(*********************************** G.D S.p.A. - Technical Department ***********************************
============= PROGRAM INFO ============
FOLDER:             TBD
MACHINES INVOLVED:  TBD 

============= DESCRIPTION =============
csp machine declaration

============= REVISIONS ===============
Date		Version	 	Author      	Description             
----------	-------		------------  	--------------------------------------------
2019/04/05 	0000.00	 	M.Grasso		Creation of the PRG

**********************************************************************************************************)
(*$R process_ref := prc; $*)
PROGRAM csp_case_feed_kinematic_tilt
VAR
		
	prc:												process;
	prc_path:											STRING;
	
	axis:												axis;
	axis_actual_position:								LREAL;
	
	fsm_enable_condition:								BOOL := FALSE;
	fsm_next_status:									csp_case_feed_kinematic_status_enum;
	fsm_status:											csp_case_feed_kinematic_status_enum;
	debug_state_machine:								BOOL := FALSE;
	debug_state_machine_one_step:						BOOL := FALSE;	
	
	in_accu_safe_pos:                                   BOOL := FALSE;
    accu_tolerance:                                     LREAL := 5.0;
    accu_safe_pos:                                      LREAL := 1334.5;
	
	cam_id:												INT := 7;

	local_test: 										BOOL := false;
END_VAR

VAR CONSTANT
	MOTOR_PHASE_VELOCITY_DEGPS:							LREAL := 8;	
	MOTOR_MAX_VELOCITY_DEGPS:							LREAL := 9600;
	MOTOR_MAX_ACCELLERATION_DEGPS2:						LREAL := 4800;
	MOTOR_MAX_DECELLERATION_DEGPS2:						LREAL := 4800;
	MOTOR_MAX_JERK_DEGPS3:								LREAL := 100000000; 
	MOTOR_MAX_FOLLOWING_ERROR_DEG:						LREAL := 2;
END_VAR

_read_var_input();

_object_manager();

IF 	NOT objects_running()
THEN
	RETURN;	
END_IF

_read_process_image();

_mode_manager();

CASE process_get_mode(prc) OF
	MODE_ABSENT,
	MODE_INACTIVE:
		RETURN;
	MODE_TEST:
		_handle_process_test();
END_CASE

_set_runtime_properties();

(********************************* BODY *********************************)

IF (axis.actual_position > (accu_safe_pos - accu_tolerance)) AND axis.actual_position < (accu_safe_pos + accu_tolerance)
THEN
	in_accu_safe_pos := TRUE;
ELSE
	in_accu_safe_pos := FALSE;   
END_IF

// Manage the accu change safe position
fsm_enable_condition := axis_is_ok(FALSE, axis)	
						AND															
						(csp_case_feed_kinematic.fsm_status = CSP_CASE_FEED_KINEMATIC_STATUS_ENABLED)
						AND
						csp_case_feed_kinematic.cartesian_mode_active
						AND							
						csp_main_accuChange.Brand_Change_Occurred;
										
IF	NOT fsm_enable_condition
	AND
	fsm_status <> CSP_CASE_FEED_KINEMATIC_STATUS_DISABLED	
THEN
	fsm_next_status	:= CSP_CASE_FEED_KINEMATIC_STATUS_DISABLED;
END_IF
					
CASE fsm_status OF
	
	CSP_CASE_FEED_KINEMATIC_STATUS_NOT_INITIALIZED:
	
        IF	axis_is_ok(return_when_absent := TRUE, CONVERSION_this := axis)
        THEN
            fsm_next_status := CSP_CASE_FEED_KINEMATIC_STATUS_DISABLED;
        END_IF
		

	CSP_CASE_FEED_KINEMATIC_STATUS_DISABLED:
	
		IF	fsm_enable_condition
			AND
			motorization_conditioner_is_execute(csp_main_services_towerLamp.buzzer_motcond) 							
		THEN	
			IF	in_accu_safe_pos
			THEN
				fsm_next_status := CSP_CASE_FEED_KINEMATIC_STATUS_CHANGE_OVER_MODE_DONE;
			ELSE								
				fsm_next_status := CSP_CASE_FEED_KINEMATIC_STATUS_ENABLED;
			END_IF
		END_IF;
		

	CSP_CASE_FEED_KINEMATIC_STATUS_ENABLED:	
	
		axis_move_absolute(
			position 		:= accu_safe_pos,
			velocity 		:= MOTOR_PHASE_VELOCITY_DEGPS,
			direction		:= AXIS_CURRENT_DIRECTION,
			acceleration 	:= MOTOR_MAX_ACCELLERATION_DEGPS2,
			deceleration 	:= MOTOR_MAX_DECELLERATION_DEGPS2,
			jerk 			:= MOTOR_MAX_JERK_DEGPS3, 
			buffer_mode 	:= AXIS_BUFFER_MODE_BUFFERED,
			CONVERSION_this := axis);
			
		IF 	axis_is_absolute_moving(axis)
		THEN
			fsm_next_status	:= CSP_CASE_FEED_KINEMATIC_STATUS_CHANGE_OVER_MODE;
		END_IF
		
		
	CSP_CASE_FEED_KINEMATIC_STATUS_CHANGE_OVER_MODE:
	
		IF 	axis_is_standstill(axis)
		THEN	
			axis_disable(axis);					
			fsm_next_status := CSP_CASE_FEED_KINEMATIC_STATUS_CHANGE_OVER_MODE_DONE;
		END_IF
		
	CSP_CASE_FEED_KINEMATIC_STATUS_CHANGE_OVER_MODE_DONE:
	
		;
		
END_CASE

IF 	NOT debug_state_machine
	OR
	debug_state_machine_one_step
THEN
	fsm_status := fsm_next_status;
	debug_state_machine_one_step := FALSE;
END_IF


(* TEMPORARY CAM CHANGE *)
IF csp_main_brand.count = '24Count'
	THEN
		cam_id := 307;
ELSIF csp_main_brand.count = '10Count'
	THEN
		cam_id := 573;
ELSIF csp_main_brand.count = '32Count'
	THEN
		cam_id := 7;
ELSIF csp_main_brand.count = '48Count'
	THEN
		cam_id := 45;
END_IF

(************************************************************************)

_handle_messages();

_write_output();

ACTION _handle_messages:
;
END_ACTION

ACTION _handle_process_test:
;
END_ACTION

ACTION _mode_manager:
IF process_mode_req_is_pending(prc)
THEN
    process_apply_mode_req_first_step(prc);
    CASE process_get_mode(prc) OF
        MODE_TO_ABSENT:
			;
        MODE_TO_INACTIVE:
			;
        MODE_TO_TEST:
			;
        MODE_TO_OPERATIONAL:
			;
    END_CASE
    process_apply_mode_req_second_step(prc);
END_IF
END_ACTION

ACTION _object_manager:
IF objects_initialization()
THEN
	sub_process_init(
		object_name					:= 'csp_case_feed_kinematic_tilt.prc', 
		process						:= csp_case_feed_kinematic.prc, 
		CONVERSION_this				:= prc);
		
	prc_path 						:= process_get_path(prc);
	
	axis_init(
		object_name					:= CONCAT(prc_path, '_axis'), 
		axis_type					:= AXIS_TYPE_VIRTUAL, 
		encoder_scaling_factor		:= G_VIRTUAL_ENCODER_SCALING_FACTOR_DEGPINC,
		modulo						:= G_NO_MODULO_DEG, 
		process						:= prc, 
		CONVERSION_this				:= axis);
	
	axis_set_max_dynamic(
		reference_velocity			:=	MOTOR_MAX_VELOCITY_DEGPS,
		velocity					:=	MOTOR_MAX_VELOCITY_DEGPS,
		acceleration				:=	MOTOR_MAX_ACCELLERATION_DEGPS2,
		deceleration				:=	MOTOR_MAX_DECELLERATION_DEGPS2,
		jerk						:=	MOTOR_MAX_JERK_DEGPS3,
		following_error				:=	MOTOR_MAX_FOLLOWING_ERROR_DEG,
		CONVERSION_this				:=	axis);
	

END_IF

IF objects_running()
THEN
	process_cycle(prc);
	axis_cycle(axis);
END_IF
END_ACTION

ACTION _read_process_image:
;
END_ACTION

ACTION _read_var_input:
;
END_ACTION

ACTION _set_runtime_properties:
axis_actual_position := axis_get_actual_incremental_position(axis);
END_ACTION

ACTION _write_output:
;
END_ACTION

END_PROGRAM

(* stored: Version 1.1.0.1, ProductVersion 3.1.4024.3
   POU csp_case_feed_kinematic_tilt: Id {89c29b54-ef12-4335-96c3-9c2a5feaefd2}, SpecialFunc None
   Action _handle_messages: Id {ca6c48f8-d046-45ae-8a13-9510e72c488c}
   Action _handle_process_test: Id {c3a03879-4e7b-4f40-a5fb-4712427e1a5b}
   Action _mode_manager: Id {518d4158-df4d-46f0-bf98-dfb82b149ad5}
   Action _object_manager: Id {b34a6487-3a6a-4110-8c55-b8ab528b8aa5}
   Action _read_process_image: Id {580df7ba-4d92-48d7-b4fb-de361185dc0f}
   Action _read_var_input: Id {db1104c9-bdd0-4b01-8726-3863f7f6aeae}
   Action _set_runtime_properties: Id {465d0da6-535d-4252-9787-800685912266}
   Action _write_output: Id {a7138920-a279-45f7-9165-61bb06ab6854} *)
